TYPE ST_Terminal_Info :
STRUCT
	
	nTerminal_State                        AT %I*			:    UINT;	// Terminal State from IO Terminal Info Data
	sTerminalInfo                                           :    STRING;
    fbTerminalInfo                                          :    FB_TerminalInfo;
END_STRUCT
END_TYPE

(* stored: Version 1.1.0.1, ProductVersion 3.1.4024.13
   DUT ST_Terminal_Info: Id {8674490a-6304-4125-8c29-3c1ed402d291} *)
